Omron CX-Programmer project 新工程 (CX-Programmer 9.72)

# PLC 新PLC1: CQM1H CPU21

## Program 新程序1 (no task)

### Section 段1

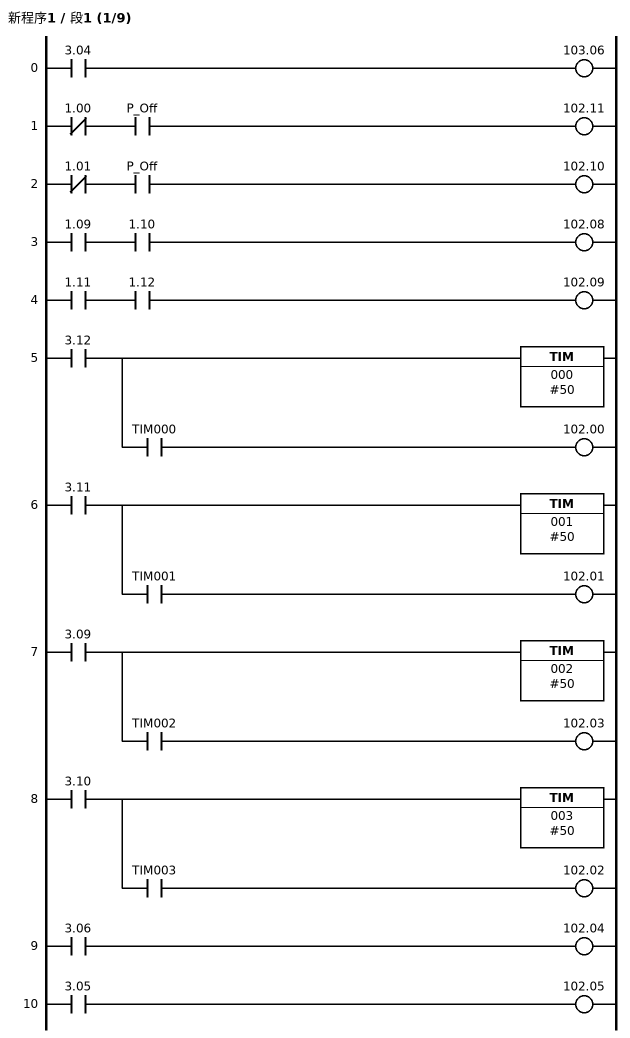
; rung 0
LD 3.04
OUT 103.06
; rung 1
LDNOT 1.00
AND P_Off
OUT 102.11
; rung 2
LDNOT 1.01
AND P_Off
OUT 102.10
; rung 3
LD 1.09
AND 1.10
OUT 102.08
; rung 4
LD 1.11
AND 1.12
OUT 102.09
; rung 5
LD 3.12
TIM 000 #50
AND TIM000
OUT 102.00
; rung 6
LD 3.11
TIM 001 #50
AND TIM001
OUT 102.01
; rung 7
LD 3.09
TIM 002 #50
AND TIM002
OUT 102.03
; rung 8
LD 3.10
TIM 003 #50
AND TIM003
OUT 102.02
; rung 9
LD 3.06
OUT 102.04
; rung 10
LD 3.05
OUT 102.05

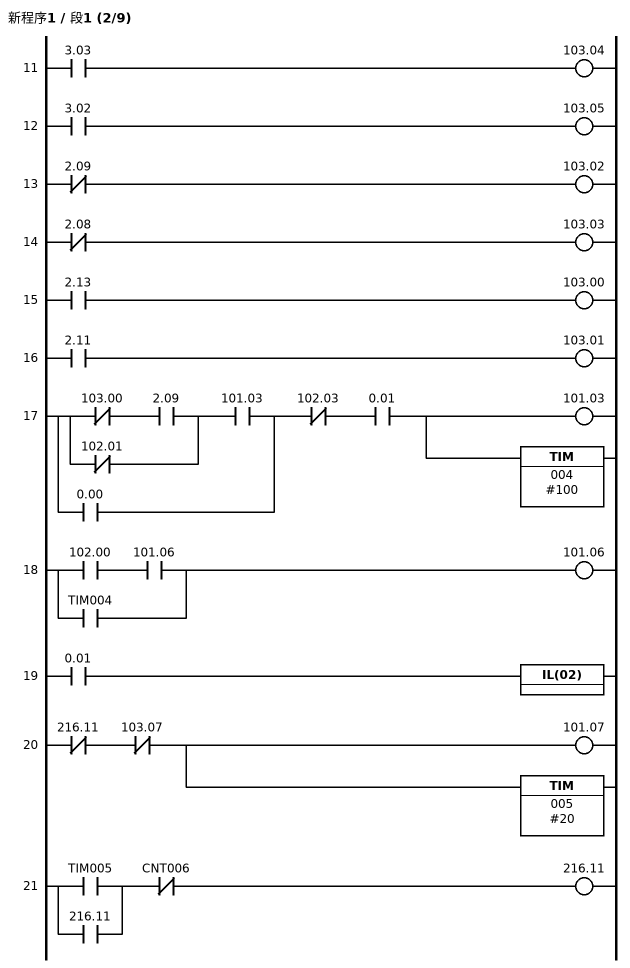
; rung 11
LD 3.03
OUT 103.04
; rung 12
LD 3.02
OUT 103.05
; rung 13
LDNOT 2.09
OUT 103.02
; rung 14
LDNOT 2.08
OUT 103.03
; rung 15
LD 2.13
OUT 103.00
; rung 16
LD 2.11
OUT 103.01
; rung 17
LDNOT 103.00
AND 2.09
ORNOT 102.01
AND 101.03
OR 0.00
ANDNOT 102.03
AND 0.01
OUT 101.03
TIM 004 #100
; rung 18
LD 102.00
AND 101.06
OR TIM004
OUT 101.06
; rung 19
LD 0.01
IL(02)
; rung 20
LDNOT 216.11
ANDNOT 103.07
OUT 101.07
TIM 005 #20
; rung 21
LD TIM005
OR 216.11
ANDNOT CNT006
OUT 216.11

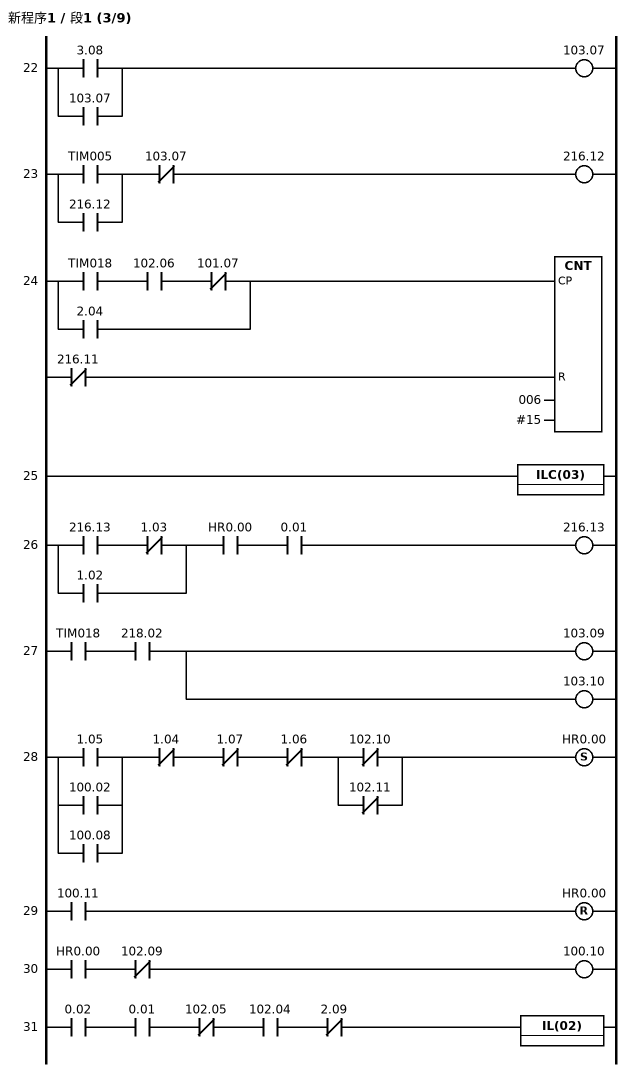
; rung 22
LD 3.08
OR 103.07
OUT 103.07
; rung 23
LD TIM005
OR 216.12
ANDNOT 103.07
OUT 216.12
; rung 24
LD TIM018
AND 102.06
ANDNOT 101.07
OR 2.04
LDNOT 216.11
CNT 006 #15
; rung 25
ILC(03)
; rung 26
LD 216.13
ANDNOT 1.03
OR 1.02
AND HR0.00
AND 0.01
OUT 216.13
; rung 27
LD TIM018
AND 218.02
OUT 103.09
OUT 103.10
; rung 28
LD 1.05
OR 100.02
OR 100.08
ANDNOT 1.04
ANDNOT 1.07
ANDNOT 1.06
LDNOT 102.10
ORNOT 102.11
ANDLD
SET HR0.00
; rung 29
LD 100.11
RSET HR0.00
; rung 30
LD HR0.00
ANDNOT 102.09
OUT 100.10
; rung 31
LD 0.02
AND 0.01
ANDNOT 102.05
AND 102.04
ANDNOT 2.09
IL(02)

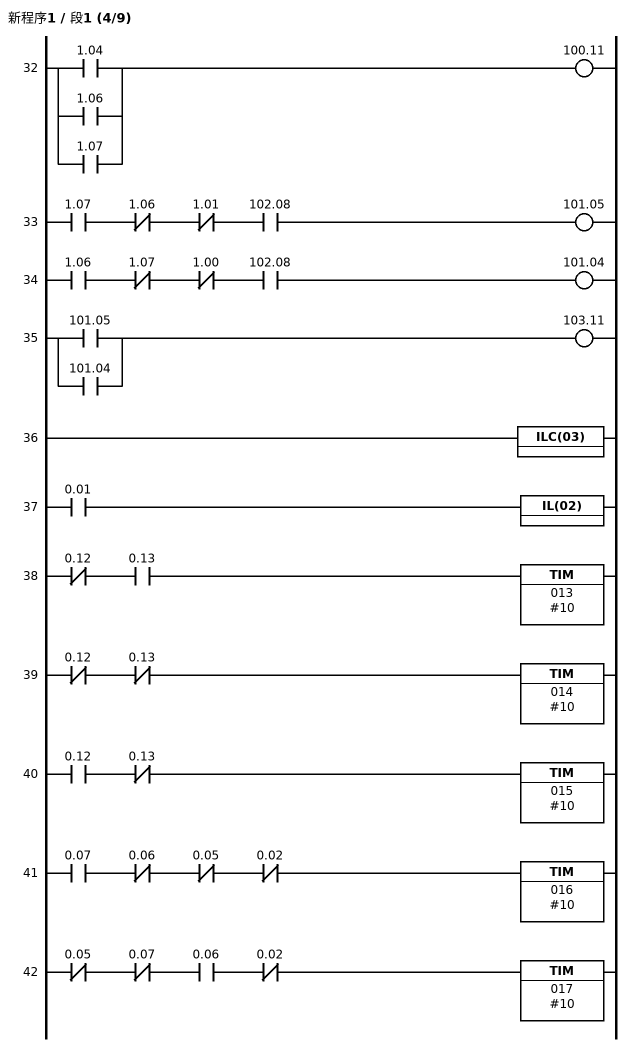
; rung 32
LD 1.04
OR 1.06
OR 1.07
OUT 100.11
; rung 33
LD 1.07
ANDNOT 1.06
ANDNOT 1.01
AND 102.08
OUT 101.05
; rung 34
LD 1.06
ANDNOT 1.07
ANDNOT 1.00
AND 102.08
OUT 101.04
; rung 35
LD 101.05
OR 101.04
OUT 103.11
; rung 36
ILC(03)
; rung 37
LD 0.01
IL(02)
; rung 38
LDNOT 0.12
AND 0.13
TIM 013 #10
; rung 39
LDNOT 0.12
ANDNOT 0.13
TIM 014 #10
; rung 40
LD 0.12
ANDNOT 0.13
TIM 015 #10
; rung 41
LD 0.07
ANDNOT 0.06
ANDNOT 0.05
ANDNOT 0.02
TIM 016 #10
; rung 42
LDNOT 0.05
ANDNOT 0.07
AND 0.06
ANDNOT 0.02
TIM 017 #10

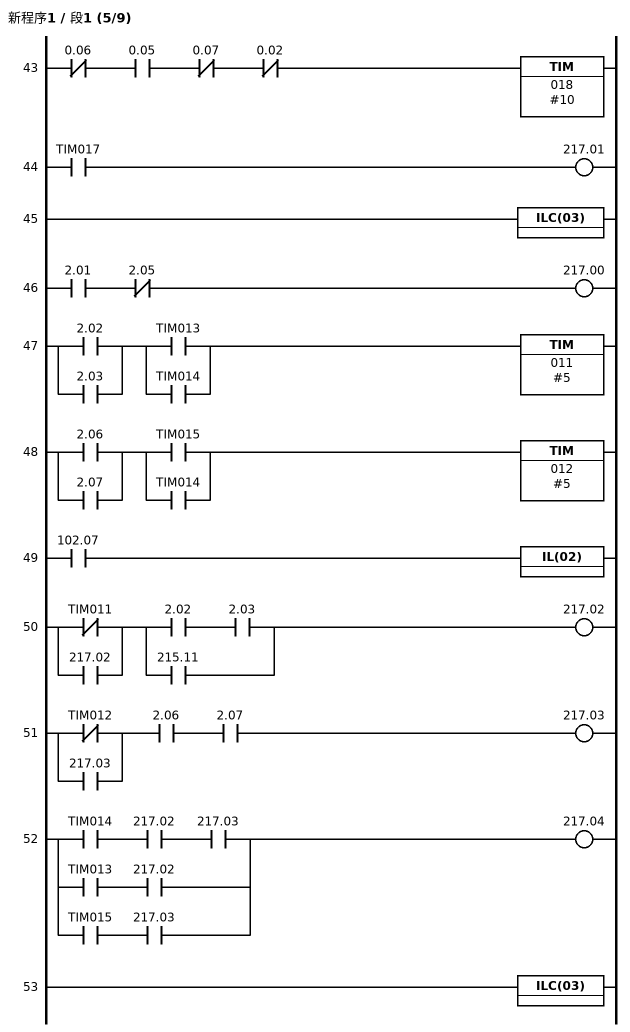
; rung 43
LDNOT 0.06
AND 0.05
ANDNOT 0.07
ANDNOT 0.02
TIM 018 #10
; rung 44
LD TIM017
OUT 217.01
; rung 45
ILC(03)
; rung 46
LD 2.01
ANDNOT 2.05
OUT 217.00
; rung 47
LD 2.02
OR 2.03
LD TIM013
OR TIM014
ANDLD
TIM 011 #5
; rung 48
LD 2.06
OR 2.07
LD TIM015
OR TIM014
ANDLD
TIM 012 #5
; rung 49
LD 102.07
IL(02)
; rung 50
LDNOT TIM011
OR 217.02
LD 2.02
AND 2.03
OR 215.11
ANDLD
OUT 217.02
; rung 51
LDNOT TIM012
OR 217.03
AND 2.06
AND 2.07
OUT 217.03
; rung 52
LD TIM014
AND 217.02
AND 217.03
LD TIM013
AND 217.02
ORLD
LD TIM015
AND 217.03
ORLD
OUT 217.04
; rung 53
ILC(03)

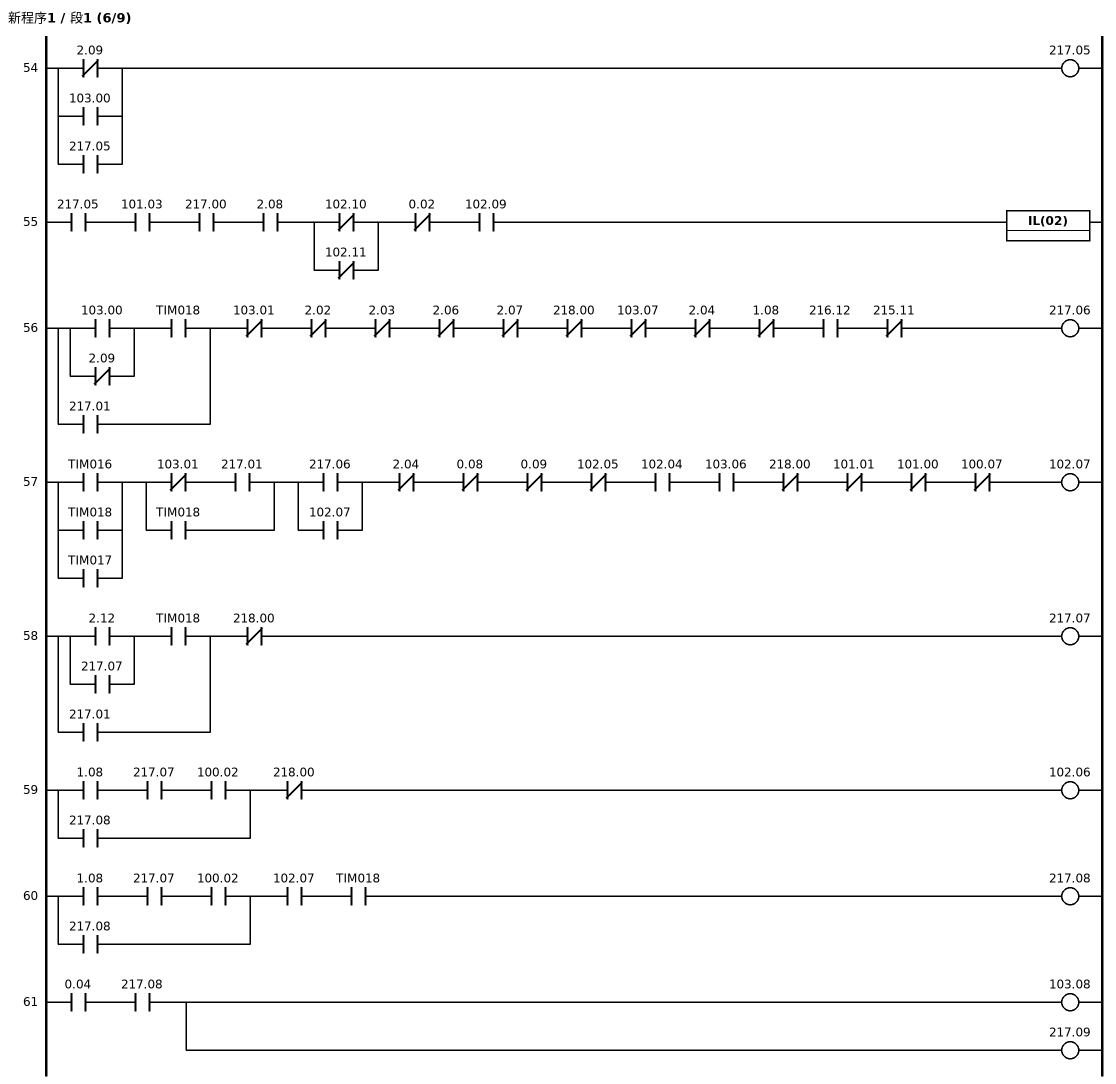
; rung 54
LDNOT 2.09
OR 103.00
OR 217.05
OUT 217.05
; rung 55
LD 217.05
AND 101.03
AND 217.00
AND 2.08
LDNOT 102.10
ORNOT 102.11
ANDLD
ANDNOT 0.02
AND 102.09
IL(02)
; rung 56
LD 103.00
ORNOT 2.09
AND TIM018
OR 217.01
ANDNOT 103.01
ANDNOT 2.02
ANDNOT 2.03
ANDNOT 2.06
ANDNOT 2.07
ANDNOT 218.00
ANDNOT 103.07
ANDNOT 2.04
ANDNOT 1.08
AND 216.12
ANDNOT 215.11
OUT 217.06
; rung 57
LD TIM016
OR TIM018
OR TIM017
LDNOT 103.01
AND 217.01
OR TIM018
ANDLD
LD 217.06
OR 102.07
ANDLD
ANDNOT 2.04
ANDNOT 0.08
ANDNOT 0.09
ANDNOT 102.05
AND 102.04
AND 103.06
ANDNOT 218.00
ANDNOT 101.01
ANDNOT 101.00
ANDNOT 100.07
OUT 102.07
; rung 58
LD 2.12
OR 217.07
AND TIM018
OR 217.01
ANDNOT 218.00
OUT 217.07
; rung 59
LD 1.08
AND 217.07
AND 100.02
OR 217.08
ANDNOT 218.00
OUT 102.06
; rung 60
LD 1.08
AND 217.07
AND 100.02
OR 217.08
AND 102.07
AND TIM018
OUT 217.08
; rung 61
LD 0.04
AND 217.08
OUT 103.08
OUT 217.09

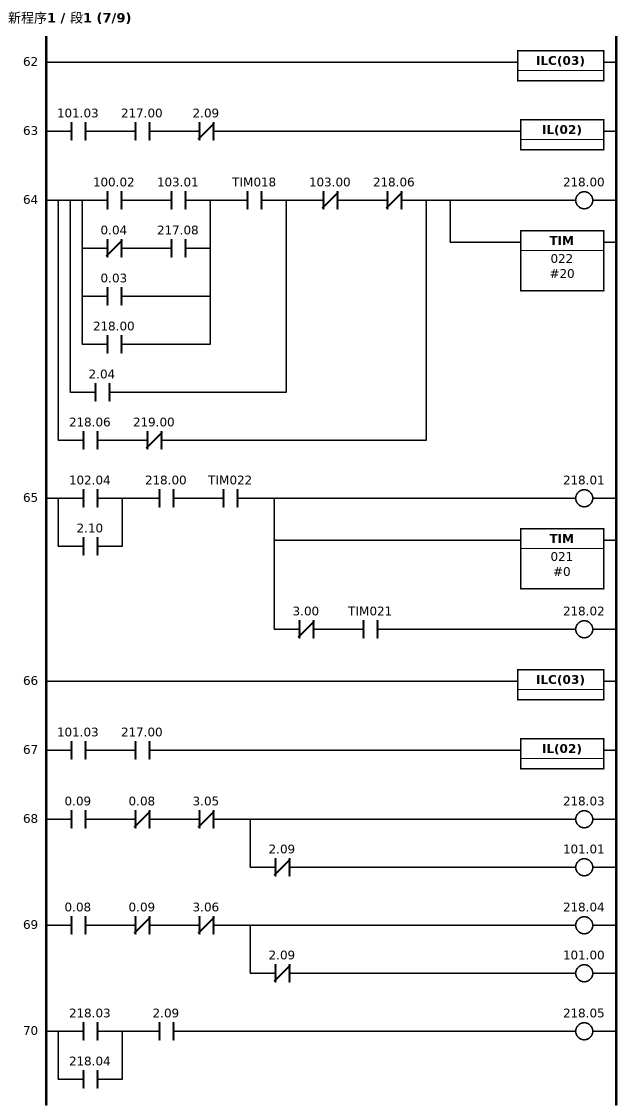
; rung 62
ILC(03)
; rung 63
LD 101.03
AND 217.00
ANDNOT 2.09
IL(02)
; rung 64
LD 100.02
AND 103.01
LDNOT 0.04
AND 217.08
ORLD
OR 0.03
OR 218.00
AND TIM018
OR 2.04
ANDNOT 103.00
ANDNOT 218.06
LD 218.06
ANDNOT 219.00
ORLD
OUT 218.00
TIM 022 #20
; rung 65
LD 102.04
OR 2.10
AND 218.00
AND TIM022
OUT 218.01
TIM 021 #0
ANDNOT 3.00
AND TIM021
OUT 218.02
; rung 66
ILC(03)
; rung 67
LD 101.03
AND 217.00
IL(02)
; rung 68
LD 0.09
ANDNOT 0.08
ANDNOT 3.05
OUT 218.03
ANDNOT 2.09
OUT 101.01
; rung 69
LD 0.08
ANDNOT 0.09
ANDNOT 3.06
OUT 218.04
ANDNOT 2.09
OUT 101.00
; rung 70
LD 218.03
OR 218.04
AND 2.09
OUT 218.05

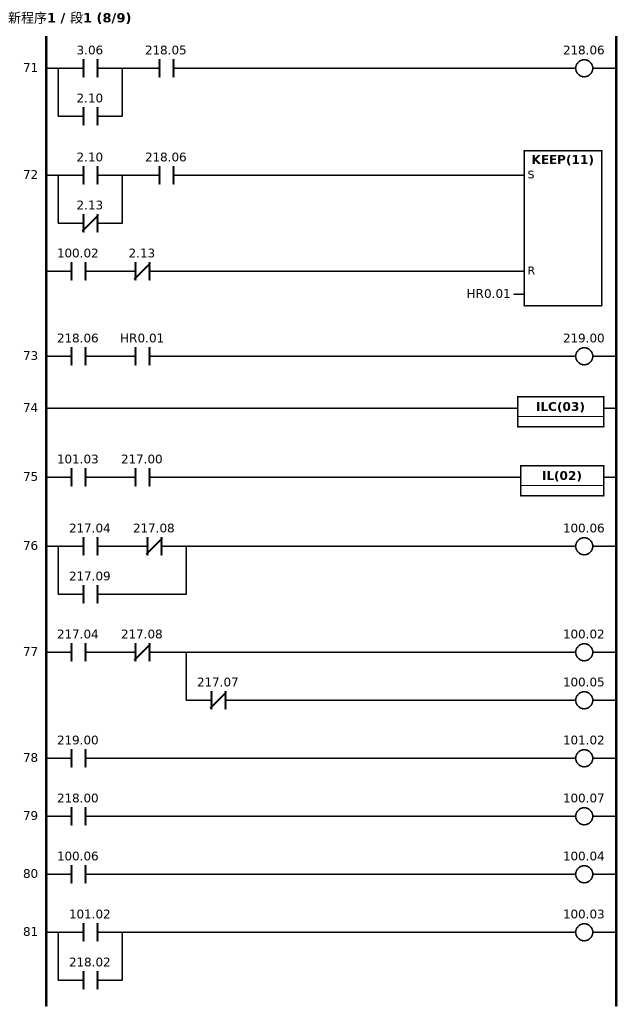
; rung 71
LD 3.06
OR 2.10
AND 218.05
OUT 218.06
; rung 72
LD 2.10
ORNOT 2.13
AND 218.06
LD 100.02
ANDNOT 2.13
KEEP(11) HR0.01
; rung 73
LD 218.06
AND HR0.01
OUT 219.00
; rung 74
ILC(03)
; rung 75
LD 101.03
AND 217.00
IL(02)
; rung 76
LD 217.04
ANDNOT 217.08
OR 217.09
OUT 100.06
; rung 77
LD 217.04
ANDNOT 217.08
OUT 100.02
ANDNOT 217.07
OUT 100.05
; rung 78
LD 219.00
OUT 101.02
; rung 79
LD 218.00
OUT 100.07
; rung 80
LD 100.06
OUT 100.04
; rung 81
LD 101.02
OR 218.02
OUT 100.03

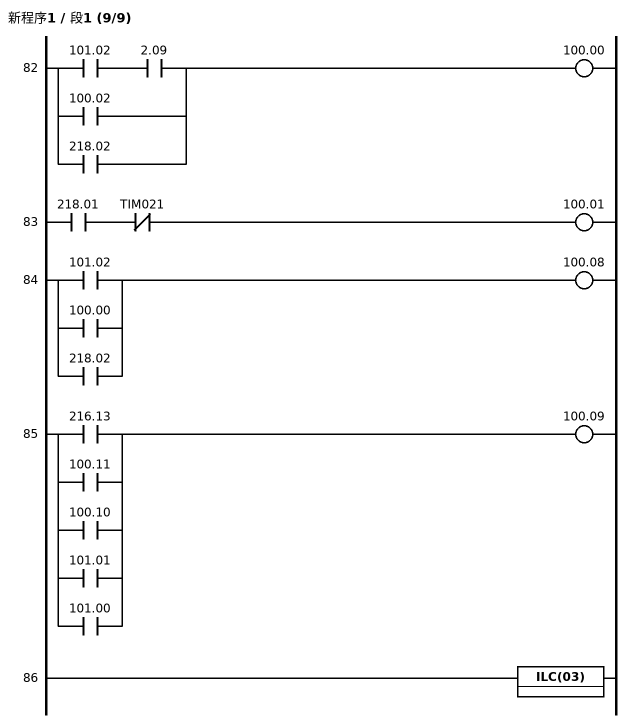
; rung 82
LD 101.02
AND 2.09
OR 100.02
OR 218.02
OUT 100.00
; rung 83
LD 218.01
ANDNOT TIM021
OUT 100.01
; rung 84
LD 101.02
OR 100.00
OR 218.02
OUT 100.08
; rung 85
LD 216.13
OR 100.11
OR 100.10
OR 101.01
OR 101.00
OUT 100.09
; rung 86
ILC(03)

### Section 段2

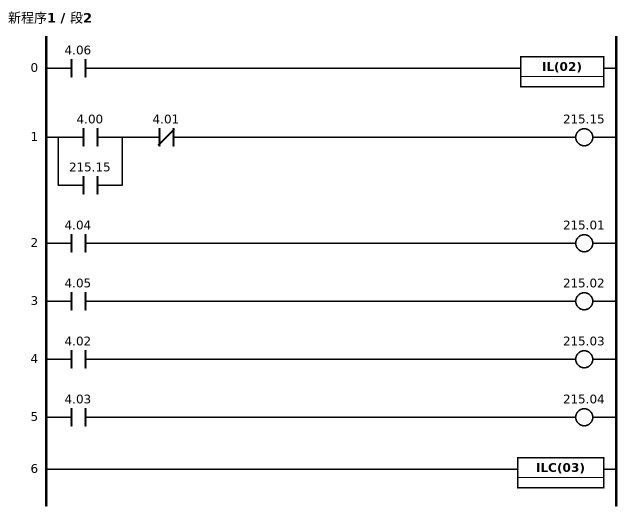
; rung 0
LD 4.06
IL(02)
; rung 1
LD 4.00
OR 215.15
ANDNOT 4.01
OUT 215.15
; rung 2
LD 4.04
OUT 215.01
; rung 3
LD 4.05
OUT 215.02
; rung 4
LD 4.02
OUT 215.03
; rung 5
LD 4.03
OUT 215.04
; rung 6
ILC(03)

### Section 段3

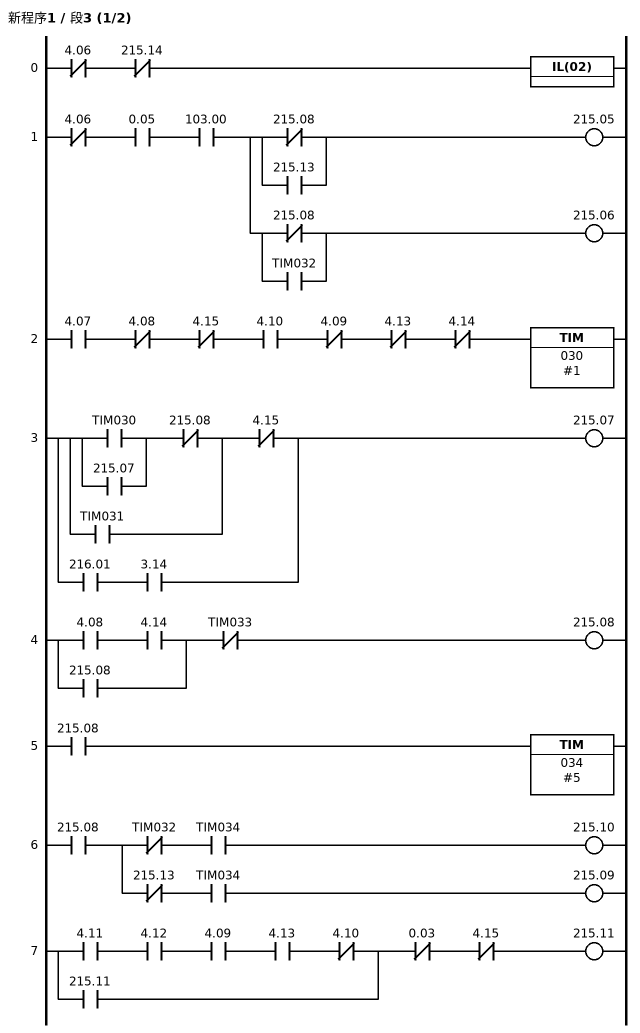
; rung 0
LDNOT 4.06
ANDNOT 215.14
IL(02)
; rung 1
LDNOT 4.06
AND 0.05
AND 103.00
OUT TR0
LDNOT 215.08
OR 215.13
ANDLD
OUT 215.05
LD TR0
LDNOT 215.08
OR TIM032
ANDLD
OUT 215.06
; rung 2
LD 4.07
ANDNOT 4.08
ANDNOT 4.15
AND 4.10
ANDNOT 4.09
ANDNOT 4.13
ANDNOT 4.14
TIM 030 #1
; rung 3
LD TIM030
OR 215.07
ANDNOT 215.08
OR TIM031
ANDNOT 4.15
LD 216.01
AND 3.14
ORLD
OUT 215.07
; rung 4
LD 4.08
AND 4.14
OR 215.08
ANDNOT TIM033
OUT 215.08
; rung 5
LD 215.08
TIM 034 #5
; rung 6
LD 215.08
OUT TR0
ANDNOT TIM032
AND TIM034
OUT 215.10
LD TR0
ANDNOT 215.13
AND TIM034
OUT 215.09
; rung 7
LD 4.11
AND 4.12
AND 4.09
AND 4.13
ANDNOT 4.10
OR 215.11
ANDNOT 0.03
ANDNOT 4.15
OUT 215.11

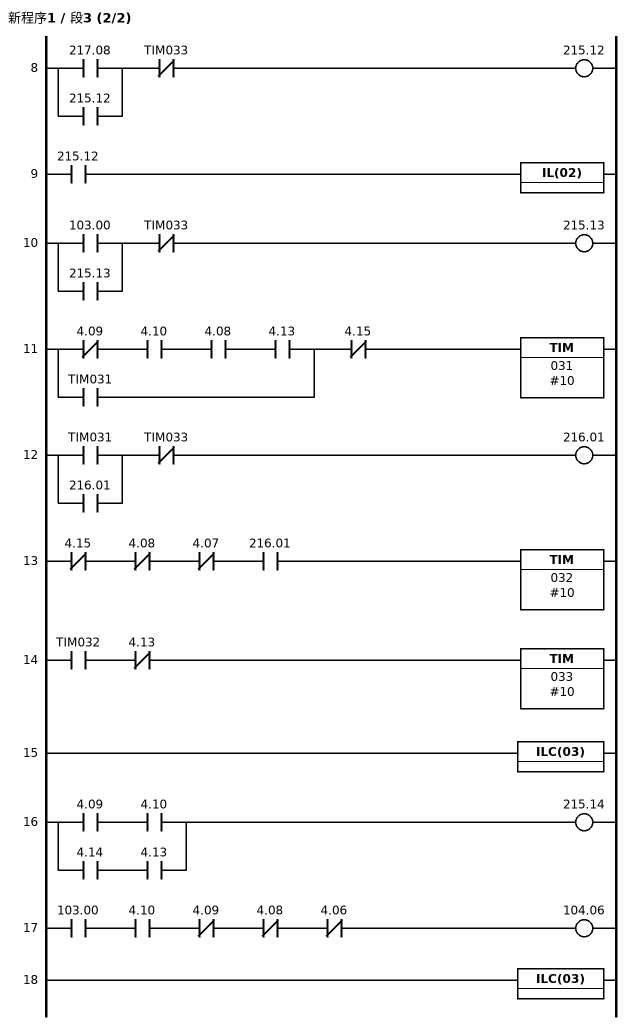
; rung 8
LD 217.08
OR 215.12
ANDNOT TIM033
OUT 215.12
; rung 9
LD 215.12
IL(02)
; rung 10
LD 103.00
OR 215.13
ANDNOT TIM033
OUT 215.13
; rung 11
LDNOT 4.09
AND 4.10
AND 4.08
AND 4.13
OR TIM031
ANDNOT 4.15
TIM 031 #10
; rung 12
LD TIM031
OR 216.01
ANDNOT TIM033
OUT 216.01
; rung 13
LDNOT 4.15
ANDNOT 4.08
ANDNOT 4.07
AND 216.01
TIM 032 #10
; rung 14
LD TIM032
ANDNOT 4.13
TIM 033 #10
; rung 15
ILC(03)
; rung 16
LD 4.09
AND 4.10
LD 4.14
AND 4.13
ORLD
OUT 215.14
; rung 17
LD 103.00
AND 4.10
ANDNOT 4.09
ANDNOT 4.08
ANDNOT 4.06
OUT 104.06
; rung 18
ILC(03)

### Section 段4

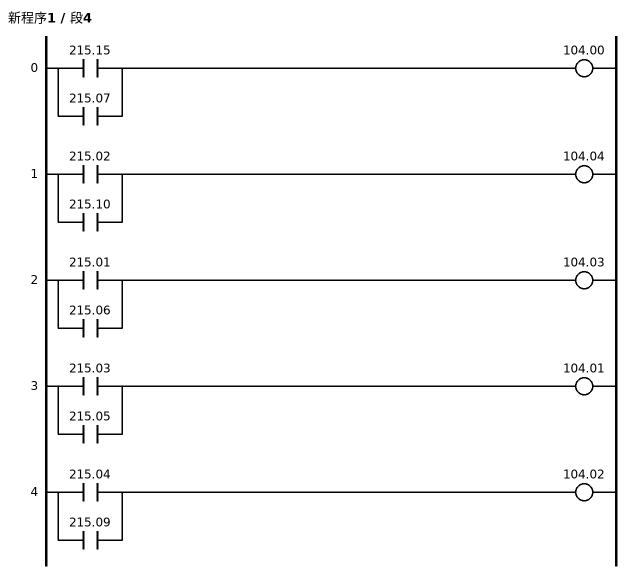
; rung 0
LD 215.15
OR 215.07
OUT 104.00
; rung 1
LD 215.02
OR 215.10
OUT 104.04
; rung 2
LD 215.01
OR 215.06
OUT 104.03
; rung 3
LD 215.03
OR 215.05
OUT 104.01
; rung 4
LD 215.04
OR 215.09
OUT 104.02

### Section 段5
; rung 0
END(01)